// TIA Portal V17 export
// export: Created 2023-05-07T12:12:11.6079197Z, ExportSetting WithDefaults, DisplayName Totally Integrated Automation Portal, DisplayVersion V17, DisplayName TIA Portal Openness, DisplayVersion V17, DisplayName TIA Portal Version Control Interface, DisplayVersion V17, DisplayName TIA Portal Test Suite Advanced, DisplayVersion V17, DisplayName STEP 7 Professional, DisplayVersion V17, DisplayName SIMATIC Energy Suite, DisplayVersion V17, DisplayName STEP 7 Safety, DisplayVersion V17, DisplayName WinCC Professional, DisplayVersion V17
ORGANIZATION_BLOCK "NeuralNetwork"   // OB31, LAD, CyclicInterrupt
TITLE = NeuralNetwork
{ S7_Optimized_Access := 'TRUE' }
VERSION : 0.1
// stored: AutoNumber true, IsIECCheckEnabled false, SetENOAutomatically false
   VAR_INPUT
      Initial_Call : Bool;   // Initial call of this OB
      Event_Count : Int;   // Events discarded
   END_VAR
   VAR_TEMP
      MV : Real;
   END_VAR
   VAR_TEMP   // added for the SCL form of the ladder/FBD networks
      _w1 : Bool;
   END_VAR
BEGIN

REGION Network 1: Call: Measurement
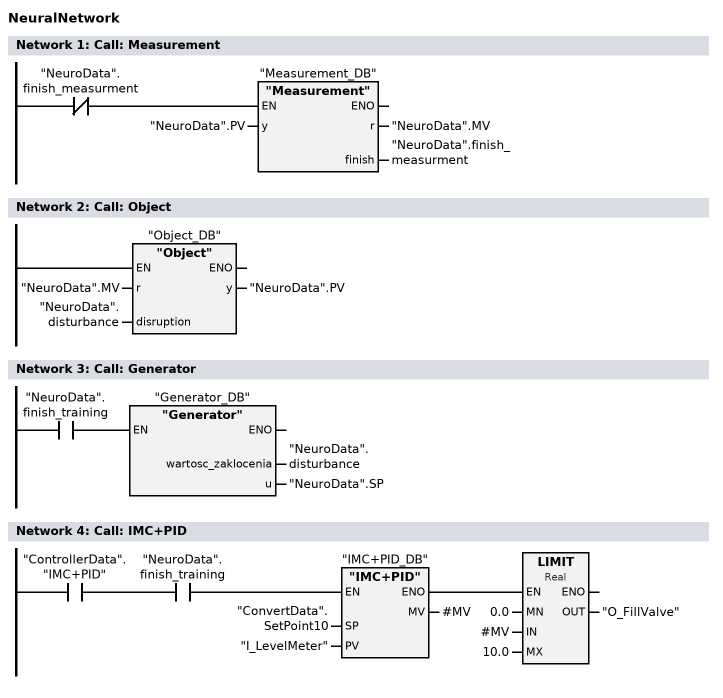
   RUNG wire#powerrail
      I_Contact( "NeuroData".finish_measurment )
      "Measurement_DB"(y := "NeuroData".PV, r => "NeuroData".MV, finish => "NeuroData".finish_measurment)
   END_RUNG
   // the same network as SCL:
   IF NOT "NeuroData".finish_measurment THEN
       "Measurement_DB"(y := "NeuroData".PV, r => "NeuroData".MV, finish => "NeuroData".finish_measurment);   // "Measurement"
   END_IF;
END_REGION

REGION Network 2: Call: Object
   RUNG wire#powerrail
      "Object_DB"(r := "NeuroData".MV, disruption := "NeuroData".disturbance, y => "NeuroData".PV)
   END_RUNG
   // the same network as SCL:
   "Object_DB"(r := "NeuroData".MV, disruption := "NeuroData".disturbance, y => "NeuroData".PV);   // "Object"
END_REGION

REGION Network 3: Call: Generator
   RUNG wire#powerrail
      Contact( "NeuroData".finish_training )
      "Generator_DB"(wartosc_zaklocenia => "NeuroData".disturbance, u => "NeuroData".SP)
   END_RUNG
   // the same network as SCL:
   IF "NeuroData".finish_training THEN
       "Generator_DB"(wartosc_zaklocenia => "NeuroData".disturbance, u => "NeuroData".SP);   // "Generator"
   END_IF;
END_REGION

REGION Network 4: Call: IMC+PID
   RUNG wire#powerrail
      Contact( "ControllerData"."IMC+PID" )
      Contact( "NeuroData".finish_training )
      "IMC+PID_DB"(SP := "ConvertData".SetPoint10, PV := "I_LevelMeter", MV => #MV)
      { S7_Templates := "value_type := Real" } Limit(mn := 0.0, in := #MV, mx := 10.0, out => "O_FillValve")
   END_RUNG
   // the same network as SCL:
   "IMC+PID_DB"(EN := "ControllerData"."IMC+PID" AND "NeuroData".finish_training,   // "IMC+PID"
                SP := "ConvertData".SetPoint10,
                PV := "I_LevelMeter",
                MV => #MV,
                ENO => #_w1);
   IF #_w1 THEN "O_FillValve" := LIMIT(MN := 0.0, IN := #MV, MX := 10.0); END_IF;
END_REGION
END_ORGANIZATION_BLOCK
